TYPE ST_AlarmEventData_TextList :
STRUCT
	qActive		: BOOL;
	diEventID	: DINT;
	iClass		: INT; 		//0 = none, 1= Maintenance, 2= Message, 3= Hint, 4= StateInfo, 5= Instruction, 6 = Warning, 7= Alarm, 8= Parameter
	sTime		: STRING;
END_STRUCT
END_TYPE

(* stored: Version 1.1.0.1
   DUT ST_AlarmEventData_TextList: Id {111e09d2-8765-453f-bd24-2e6547cfbff8} *)
